// TIA Portal V16 export
// export: Created 2021-07-12T14:47:18.2764165Z, ExportSetting WithDefaults, DisplayName Totally Integrated Automation Portal, DisplayVersion V16, DisplayName TIA Portal Version Control Interface, DisplayVersion V16, DisplayName TIA Portal Openness, DisplayVersion V16, DisplayName STEP 7 Professional, DisplayVersion V16, DisplayName STEP 7 Safety, DisplayVersion V16, DisplayName WinCC Professional, DisplayVersion V16
TYPE "LSimaHydTO_typeVCharData"
TITLE = LSimaHydTO_typeVCharData
// Valve characteristic description
// stored: IsFailsafeCompliant false
   STRUCT
      QOutput { S7_SetPoint := 'True'} : Array[0.."LSIMAHYD_VCHAR_POINTS_UPPER_LIMIT"] of Real;   // Output values array
      Velocity { S7_SetPoint := 'True'} : Array[0.."LSIMAHYD_VCHAR_POINTS_UPPER_LIMIT"] of Real;   // Velocity values array
      VelocityLimitPositive { S7_SetPoint := 'True'} : Real;   // Max velocity in positive direction
      VelocityLimitNegative { S7_SetPoint := 'True'} : Real;   // Max velocity in negative direction
      ZeroZonePositive { S7_SetPoint := 'True'} : Real;   // Overlapping zone of valve in positive direction
      ZeroZoneNegative { S7_SetPoint := 'True'} : Real;   // Overlapping zone of valve in negative direction
      MaxIdx { S7_SetPoint := 'True'} : Int;   // Max used index in arrays
      "Name" { S7_SetPoint := 'True'} : WString[24];   // Symbolic name displayed on HMI for index of array
   END_STRUCT;
END_TYPE
